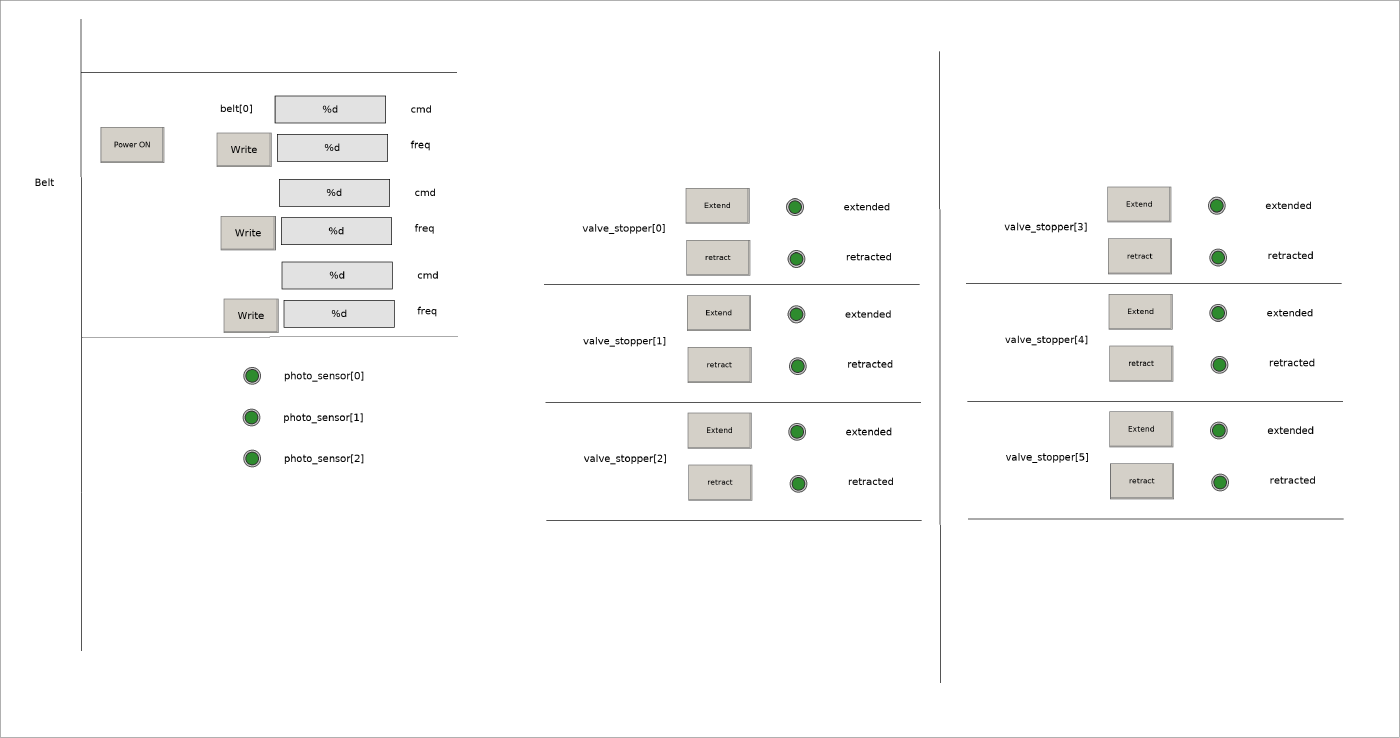
VISUALIZATION v_LB  // 2048x1080
VAR_IN_OUT
	dIO_LB		: LateralBuf_Module;
END_VAR
    Line (118,28) (119,952)
    Line (119,106) (668,106)
    Label (833,321 160x26), "valve_stopper[0]"
    Button (1003,275 93x52), "Extend", colour toggle: dIO_LB.valve_stopper[0].extend
        OnMouseDown: execute { dIO_LB.valve_stopper[0].extend := TRUE; dIO_LB.valve_stopper[0].retract := FALSE; }
    Button (1004,351 93x52), "retract", colour toggle: dIO_LB.valve_stopper[0].retract
        OnMouseDown: execute { dIO_LB.valve_stopper[0].extend := FALSE; dIO_LB.valve_stopper[0].retract := TRUE; }
    Lamp1 (1148,288 30x30), variable: dIO_LB.valve_stopper[0].extended, style: Lamp-Lamp1-Green
    Lamp1 (1150,364 30x30), variable: dIO_LB.valve_stopper[0].retracted, style: Lamp-Lamp1-Green
    Label (1202,290 132x26), "extended"
    Label (1205,363 132x26), "retracted"
    Label (834,486 160x26), "valve_stopper[1]"
    Line (796,416) (1345,416)
    Line (798,589) (1347,589)
    Rectangle (402,140 162x40), "%d", text variable: dIO_LB.belt[0].fbconverter.cmd
        OnMouseClick: write the text variable via Default
    Rectangle (405,196 162x40), "%d", text variable: dIO_LB.belt[0].fbconverter.freq
        OnMouseClick: write the text variable via Default
    Label (280,146 132x26), "belt[0]"
    Label (550,147 132x26), "cmd"
    Label (549,199 132x26), "freq"
    Button (147,186 93x52), "Power ON", colour toggle: dIO_LB.power_beltConv
        toggle dIO_LB.power_beltConv
    Button (317,194 80x50), "Write"
        OnMouseDown: execute { dIO_LB.belt[0].fbconverter.bSetParaEx	:= TRUE; }
        OnMouseUp: execute { dIO_LB.belt[0].fbconverter.bSetParaEx	:= FALSE; }
    Lamp1 (354,535 30x30), variable: dIO_LB.photo_sensor[0], style: Lamp-Lamp1-Green
    Label (408,537 132x26), "photo_sensor[0]"
    Lamp1 (353,596 30x30), variable: dIO_LB.photo_sensor[1], style: Lamp-Lamp1-Green
    Label (407,598 132x26), "photo_sensor[1]"
    Lamp1 (354,656 30x30), variable: dIO_LB.photo_sensor[2], style: Lamp-Lamp1-Green
    Label (408,658 132x26), "photo_sensor[2]"
    Line (120,493) (669,492)
    Label (25,254 80x26), "Belt"
    Button (1005,432 93x52), "Extend", colour toggle: dIO_LB.valve_stopper[1].extend
        OnMouseDown: execute { dIO_LB.valve_stopper[1].extend := TRUE; dIO_LB.valve_stopper[1].retract := FALSE; }
    Button (1006,508 93x52), "retract", colour toggle: dIO_LB.valve_stopper[1].retract
        OnMouseDown: execute { dIO_LB.valve_stopper[1].extend := FALSE; dIO_LB.valve_stopper[1].retract := TRUE; }
    Lamp1 (1150,445 30x30), variable: dIO_LB.valve_stopper[1].extended, style: Lamp-Lamp1-Green
    Lamp1 (1152,521 30x30), variable: dIO_LB.valve_stopper[1].retracted, style: Lamp-Lamp1-Green
    Label (1204,447 132x26), "extended"
    Label (1207,520 132x26), "retracted"
    Rectangle (408,262 162x40), "%d", text variable: dIO_LB.belt[1].fbconverter.cmd
        OnMouseClick: write the text variable via Default
    Rectangle (411,318 162x40), "%d", text variable: dIO_LB.belt[1].fbconverter.freq
        OnMouseClick: write the text variable via Default
    Label (556,269 132x26), "cmd"
    Label (555,321 132x26), "freq"
    Button (323,316 80x50), "Write"
        OnMouseDown: execute { dIO_LB.belt[1].fbconverter.bSetParaEx	:= TRUE; }
        OnMouseUp: execute { dIO_LB.belt[1].fbconverter.bSetParaEx	:= FALSE; }
    Rectangle (412,383 162x40), "%d", text variable: dIO_LB.belt[2].fbconverter.cmd
        OnMouseClick: write the text variable via Default
    Rectangle (415,439 162x40), "%d", text variable: dIO_LB.belt[2].fbconverter.freq
        OnMouseClick: write the text variable via Default
    Label (560,390 132x26), "cmd"
    Label (559,442 132x26), "freq"
    Button (327,437 80x50), "Write"
        OnMouseDown: execute { dIO_LB.belt[2].fbconverter.bSetParaEx	:= TRUE; }
        OnMouseUp: execute { dIO_LB.belt[2].fbconverter.bSetParaEx	:= FALSE; }
    Label (835,658 160x26), "valve_stopper[2]"
    Line (799,761) (1348,761)
    Button (1006,604 93x52), "Extend", colour toggle: dIO_LB.valve_stopper[2].extend
        OnMouseDown: execute { dIO_LB.valve_stopper[2].extend := TRUE; dIO_LB.valve_stopper[2].retract := FALSE; }
    Button (1007,680 93x52), "retract", colour toggle: dIO_LB.valve_stopper[2].retract
        OnMouseDown: execute { dIO_LB.valve_stopper[2].extend := FALSE; dIO_LB.valve_stopper[2].retract := TRUE; }
    Lamp1 (1151,617 30x30), variable: dIO_LB.valve_stopper[2].extended, style: Lamp-Lamp1-Green
    Lamp1 (1153,693 30x30), variable: dIO_LB.valve_stopper[2].retracted, style: Lamp-Lamp1-Green
    Label (1205,619 132x26), "extended"
    Label (1208,692 132x26), "retracted"
    Label (1450,319 160x26), "valve_stopper[3]"
    Button (1620,273 93x52), "Extend", colour toggle: dIO_LB.valve_stopper[3].extend
        OnMouseDown: execute { dIO_LB.valve_stopper[3].extend := TRUE; dIO_LB.valve_stopper[3].retract := FALSE; }
    Button (1621,349 93x52), "retract", colour toggle: dIO_LB.valve_stopper[3].retract
        OnMouseDown: execute { dIO_LB.valve_stopper[3].extend := FALSE; dIO_LB.valve_stopper[3].retract := TRUE; }
    Lamp1 (1765,286 30x30), variable: dIO_LB.valve_stopper[3].extended, style: Lamp-Lamp1-Green
    Lamp1 (1767,362 30x30), variable: dIO_LB.valve_stopper[3].retracted, style: Lamp-Lamp1-Green
    Label (1819,288 132x26), "extended"
    Label (1822,361 132x26), "retracted"
    Label (1451,484 160x26), "valve_stopper[4]"
    Line (1413,414) (1962,414)
    Line (1415,587) (1964,587)
    Button (1622,430 93x52), "Extend", colour toggle: dIO_LB.valve_stopper[4].extend
        OnMouseDown: execute { dIO_LB.valve_stopper[4].extend := TRUE; dIO_LB.valve_stopper[4].retract := FALSE; }
    Button (1623,506 93x52), "retract", colour toggle: dIO_LB.valve_stopper[4].retract
        OnMouseDown: execute { dIO_LB.valve_stopper[4].extend := FALSE; dIO_LB.valve_stopper[4].retract := TRUE; }
    Lamp1 (1767,443 30x30), variable: dIO_LB.valve_stopper[4].extended, style: Lamp-Lamp1-Green
    Lamp1 (1769,519 30x30), variable: dIO_LB.valve_stopper[4].retracted, style: Lamp-Lamp1-Green
    Label (1821,445 132x26), "extended"
    Label (1824,518 132x26), "retracted"
    Label (1452,656 160x26), "valve_stopper[5]"
    Line (1416,759) (1965,759)
    Button (1623,602 93x52), "Extend", colour toggle: dIO_LB.valve_stopper[5].extend
        OnMouseDown: execute { dIO_LB.valve_stopper[5].extend := TRUE; dIO_LB.valve_stopper[5].retract := FALSE; }
    Button (1624,678 93x52), "retract", colour toggle: dIO_LB.valve_stopper[5].retract
        OnMouseDown: execute { dIO_LB.valve_stopper[5].extend := FALSE; dIO_LB.valve_stopper[5].retract := TRUE; }
    Lamp1 (1768,615 30x30), variable: dIO_LB.valve_stopper[5].extended, style: Lamp-Lamp1-Green
    Lamp1 (1770,691 30x30), variable: dIO_LB.valve_stopper[5].retracted, style: Lamp-Lamp1-Green
    Label (1822,617 132x26), "extended"
    Label (1825,690 132x26), "retracted"
    Line (1374,75) (1375,999)
END_VISUALIZATION

(* stored: Version 1.1.0.1, ProductVersion 3.1.4024.12
   Visu v_LB: Id {16aaa72a-8456-4877-947b-3376f7331b28} *)
